// TIA Portal V20 export
DATA_BLOCK "GLOBAL_HMI_SCREEN_NO_IF_DB"   // DB206
{ S7_Optimized_Access := 'TRUE' }
// stored: AutoNumber false, MemoryReserve 100
   VAR
      HMI : Array[0..1] of "HMI_SCREEN_NO_AREA_POINTER_UDT";
   END_VAR
BEGIN
END_DATA_BLOCK
